(* PLC project Controller_Project, Sphere_UseCases Controller_Project 1.0 *)
(* stored: creationDateTime 2025-09-25T18:23:17, modificationDateTime 2025-09-25T18:23:17 *)

TYPE HMI_UDT : STRUCT
  Start_PB : BOOL;
  Stop_PB : BOOL;
  Start_Active : BOOL;
  Stop_Active : BOOL;
END_STRUCT;
END_TYPE

TYPE P1_UDT : STRUCT
  RW_Tank_tnk_lvl : REAL;
  RW_Pump_flow : REAL;
  RW_Tank_PR_Valve_sts : BOOL;
  RW_Tank_P6B_Valve_sts : BOOL;
  RW_Tank_P_Valve_sts : BOOL;
  RW_Pump_sts : BOOL;
  RW_Pump_fault : BOOL;
  RW_Pump : REAL;
  RW_Tank_PR_Valve : BOOL;
  RW_Tank_P_Valve : BOOL;
  RW_Pump_start : BOOL;
  RW_Pump_stop : BOOL;
  RW_Tank_P6B_Valve : BOOL;
END_STRUCT;
END_TYPE

TYPE P2_UDT : STRUCT
  ChemTreat_NaCl_Tank_tnk_lvl : REAL;
  ChemTreat_NaOCl_Tank_tnk_lvl : REAL;
  ChemTreat_HCl_Tank_tnk_lvl : REAL;
  ChemTreat_NaCl_Tank_Valve_sts : BOOL;
  ChemTreat_NaOCl_Tank_Valve_sts : BOOL;
  ChemTreat_HCl_Tank_Valve_sts : BOOL;
  ChemTreat_NaCl_Tank_Valve : BOOL;
  ChemTreat_NaOCl_Tank_Valve : BOOL;
  ChemTreat_HCl_Tank_Valve : BOOL;
END_STRUCT;
END_TYPE

TYPE P3_UDT : STRUCT
  Ultrafiltration_UFFT_Tank_tnk_lvl : REAL;
  Ultrafiltration_UFFT_Tank_Valve_sts : BOOL;
  Ultrafiltration_UF_Drain_Valve_sts : BOOL;
  Ultrafiltration_UF_ROFT_Valve_sts : BOOL;
  Ultrafiltration_UF_BWP_Valve_sts : BOOL;
  Ultrafiltration_UFFT_Tank_Valve : BOOL;
  Ultrafiltration_UF_Drain_Valve : BOOL;
  Ultrafiltration_UF_ROFT_Valve : BOOL;
  Ultrafiltration_UF_BWP_Valve : BOOL;
END_STRUCT;
END_TYPE

TYPE Phases_UDT : STRUCT
  Filling : BOOL;
  Draining : BOOL;
END_STRUCT;
END_TYPE

TYPE RW_tank_AL_UDT : STRUCT
  LL_alarm : BOOL;
  L_alarm : BOOL;
  H_alarm : BOOL;
  HH_alarm : BOOL;
END_STRUCT;
END_TYPE

TYPE System_State_UDT : STRUCT
  IDLE : BOOL;
  START : BOOL;
  RUNNING : BOOL;
  SHUTDOWN : BOOL;
  Permissives : ARRAY[0..31] OF BOOL;
  Permissives_Ready : BOOL;
END_STRUCT;
END_TYPE

TYPE SYS_MESSAGES : STRUCT
  ProgramScanTime : DINT;
  AvailableMemory : REAL;
  ControllerStatus : SINT;
  ScanTime : REAL;
END_STRUCT;
END_TYPE

PROGRAM MainProgram
  VAR_INPUT
    dbg_Alarms_ZZZZZZZZZZRW_tank_AL0 : SINT;
    dbg_Alarms_LL_alarm : BOOL;
    dbg_Alarms_L_alarm : BOOL;
    dbg_Alarms_H_alarm : BOOL;
    dbg_Alarms_HH_alarm : BOOL;
    dbg_GSV_Message_ProgramScanTime : DINT;
    dbg_GSV_Message_AvailableMemory : REAL;
    dbg_GSV_Message_ControllerStatus : SINT;
    dbg_GSV_Message_ScanTime : REAL;
    dbg_HMI_ZZZZZZZZZZUDT0 : SINT;
    dbg_HMI_Start_PB : BOOL;
    dbg_HMI_Stop_PB : BOOL;
    dbg_HMI_Start_Active : BOOL;
    dbg_HMI_Stop_Active : BOOL;
    dbg_P1_RW_Tank_tnk_lvl : REAL;
    dbg_P1_RW_Pump_flow : REAL;
    dbg_P1_ZZZZZZZZZZP1_UDT2 : SINT;
    dbg_P1_RW_Tank_PR_Valve_sts : BOOL;
    dbg_P1_RW_Tank_P6B_Valve_sts : BOOL;
    dbg_P1_RW_Tank_P_Valve_sts : BOOL;
    dbg_P1_RW_Pump_sts : BOOL;
    dbg_P1_RW_Pump_fault : BOOL;
    dbg_P1_RW_Pump : REAL;
    dbg_P1_ZZZZZZZZZZP1_UDT9 : SINT;
    dbg_P1_RW_Tank_PR_Valve : BOOL;
    dbg_P1_RW_Tank_P_Valve : BOOL;
    dbg_P1_RW_Pump_start : BOOL;
    dbg_P1_RW_Pump_stop : BOOL;
    dbg_P1_RW_Tank_P6B_Valve : BOOL;
    dbg_P1_SYS_ZZZZZZZZZZSystem_Sta0 : SINT;
    dbg_P1_SYS_IDLE : BOOL;
    dbg_P1_SYS_START : BOOL;
    dbg_P1_SYS_RUNNING : BOOL;
    dbg_P1_SYS_SHUTDOWN : BOOL;
    dbg_P1_SYS_Permissives : ARRAY[0..31] OF BOOL;
    dbg_P1_SYS_ZZZZZZZZZZSystem_Sta6 : SINT;
    dbg_P1_SYS_Permissives_Ready : BOOL;
    dbg_P2_ChemTreat_NaCl_Tank_tnk_lvl : REAL;
    dbg_P2_ChemTreat_NaOCl_Tank_tnk_lvl : REAL;
    dbg_P2_ChemTreat_HCl_Tank_tnk_lvl : REAL;
    dbg_P2_ZZZZZZZZZZP2_UDT3 : SINT;
    dbg_P2_ChemTreat_NaCl_Tank_Valve_sts : BOOL;
    dbg_P2_ChemTreat_NaOCl_Tank_Valve_sts : BOOL;
    dbg_P2_ChemTreat_HCl_Tank_Valve_sts : BOOL;
    dbg_P2_ChemTreat_NaCl_Tank_Valve : BOOL;
    dbg_P2_ChemTreat_NaOCl_Tank_Valve : BOOL;
    dbg_P2_ChemTreat_HCl_Tank_Valve : BOOL;
    dbg_P3_Ultrafiltration_UFFT_Tank_tnk_lvl : REAL;
    dbg_P3_ZZZZZZZZZZP3_UDT1 : SINT;
    dbg_P3_Ultrafiltration_UFFT_Tank_Valve_sts : BOOL;
    dbg_P3_Ultrafiltration_UF_Drain_Valve_sts : BOOL;
    dbg_P3_Ultrafiltration_UF_ROFT_Valve_sts : BOOL;
    dbg_P3_Ultrafiltration_UF_BWP_Valve_sts : BOOL;
    dbg_P3_Ultrafiltration_UFFT_Tank_Valve : BOOL;
    dbg_P3_Ultrafiltration_UF_Drain_Valve : BOOL;
    dbg_P3_Ultrafiltration_UF_ROFT_Valve : BOOL;
    dbg_P3_Ultrafiltration_UF_BWP_Valve : BOOL;
    di_2_0 AT %IX2.0 : BOOL;
    di_2_1 AT %IX2.1 : BOOL;
    di_2_10 AT %IX2.10 : BOOL;
    di_2_11 AT %IX2.11 : BOOL;
    di_2_2 AT %IX2.2 : BOOL;
    di_2_3 AT %IX2.3 : BOOL;
    di_2_4 AT %IX2.4 : BOOL;
    di_2_5 AT %IX2.5 : BOOL;
    di_2_6 AT %IX2.6 : BOOL;
    di_2_8 AT %IX2.8 : BOOL;
    di_2_9 AT %IX2.9 : BOOL;
    ai_7_0 AT %IW70 : REAL;
    di_7_ch0halarm AT %IX7.0 : BOOL;
    di_7_ch0hhalarm AT %IX7.0 : BOOL;
    di_7_ch0lalarm AT %IX7.0 : BOOL;
    di_7_ch0llalarm AT %IX7.0 : BOOL;
    ai_7_1 AT %IW71 : REAL;
    ai_7_2 AT %IW72 : REAL;
    ai_7_3 AT %IW73 : REAL;
    ai_7_4 AT %IW74 : REAL;
    ai_7_5 AT %IW75 : REAL;
  END_VAR
  VAR_OUTPUT
    ao_10_0 AT %QW100 : REAL;
    do_5_0 AT %QX5.0 : BOOL;
    do_5_1 AT %QX5.1 : BOOL;
    do_5_10 AT %QX5.10 : BOOL;
    do_5_11 AT %QX5.11 : BOOL;
    do_5_2 AT %QX5.2 : BOOL;
    do_5_3 AT %QX5.3 : BOOL;
    do_5_4 AT %QX5.4 : BOOL;
    do_5_5 AT %QX5.5 : BOOL;
    do_5_6 AT %QX5.6 : BOOL;
    do_5_7 AT %QX5.7 : BOOL;
    do_5_8 AT %QX5.8 : BOOL;
    do_5_9 AT %QX5.9 : BOOL;
  END_VAR

            (* IO_setup *)
(* P1 Analog Input *)
dbg_P1_RW_Tank_tnk_lvl := ai_7_0;
dbg_P1_RW_Pump_flow := ai_7_1;
(* P1 Digital Input *)
dbg_P1_RW_Tank_PR_Valve_sts := di_2_0;
dbg_P1_RW_Tank_P6B_Valve_sts := di_2_1;
dbg_P1_RW_Tank_P_Valve_sts := di_2_2;
dbg_P1_RW_Pump_sts := di_2_3;
dbg_P1_RW_Pump_fault := di_2_4;
(* P1 Analog Output *)
dbg_P1_RW_Pump := ao_10_0;
(* Digital Output *)
dbg_P1_RW_Tank_PR_Valve := do_5_0;
dbg_P1_RW_Tank_P6B_Valve := do_5_1;
dbg_P1_RW_Tank_P_Valve := do_5_2;
dbg_P1_RW_Pump_start := do_5_3;
dbg_P1_RW_Pump_stop := do_5_4;
(* P1 raw water tank alarms *)
dbg_Alarms_LL_alarm := di_7_ch0llalarm;
dbg_Alarms_L_alarm := di_7_ch0lalarm;
dbg_Alarms_H_alarm := di_7_ch0halarm;
dbg_Alarms_HH_alarm := di_7_ch0hhalarm;
(* P2 Analog Input *)
dbg_P2_ChemTreat_NaCl_Tank_tnk_lvl := ai_7_2;
dbg_P2_ChemTreat_NaOCl_Tank_tnk_lvl := ai_7_3;
dbg_P2_ChemTreat_HCl_Tank_tnk_lvl := ai_7_4;
(* P2 Digital Input *)
dbg_P2_ChemTreat_NaCl_Tank_Valve_sts := di_2_5;
dbg_P2_ChemTreat_NaOCl_Tank_Valve_sts := di_2_6;
(* P2 Analog Output *)
(* NONE *)
(* P2 Digital Output *)
dbg_P2_ChemTreat_NaCl_Tank_Valve := do_5_5;
dbg_P2_ChemTreat_NaOCl_Tank_Valve := do_5_6;
dbg_P2_ChemTreat_HCl_Tank_Valve := do_5_7;
(* P3 Analog Input *)
dbg_P3_Ultrafiltration_UFFT_Tank_tnk_lvl := ai_7_5;
(* P3 Digital Input *)
dbg_P3_Ultrafiltration_UFFT_Tank_Valve_sts := di_2_8;
dbg_P3_Ultrafiltration_UF_Drain_Valve_sts := di_2_9;
dbg_P3_Ultrafiltration_UF_Drain_Valve_sts := di_2_10;
dbg_P3_Ultrafiltration_UF_BWP_Valve_sts := di_2_11;
(* P3 Analog Output *)
(* none *)
(* P3 Digital Output *)
dbg_P3_Ultrafiltration_UFFT_Tank_Valve := do_5_8;
dbg_P3_Ultrafiltration_UF_Drain_Valve := do_5_9;
dbg_P3_Ultrafiltration_UF_ROFT_Valve := do_5_10;
dbg_P3_Ultrafiltration_UF_BWP_Valve := do_5_11;

(* Raw_water_control *)
if dbg_P1_RW_Tank_tnk_lvl = 250.0 and dbg_P1_SYS_RUNNING then
dbg_P1_RW_Pump_stop := True;
dbg_P1_RW_Pump_start := False; (* send the outputs *)
dbg_Alarms_LL_alarm := True;
(* if the level is at 500 or lower than 500 open the valve *)
elsif dbg_P1_RW_Tank_tnk_lvl <= 500.0 and dbg_P1_SYS_RUNNING then
(* output to turn the valve open *)
dbg_P1_RW_Tank_PR_Valve := True;
dbg_Alarms_L_alarm := True;
(* if level is at 800 *)
elsif  dbg_P1_RW_Tank_tnk_lvl = 800.0 and dbg_P1_SYS_RUNNING then
dbg_P1_RW_Tank_PR_Valve := False; (* close the valve *)
dbg_Alarms_H_alarm := True;
elsif dbg_P1_RW_Tank_tnk_lvl = 1200.0 and dbg_P1_SYS_RUNNING then
dbg_Alarms_HH_alarm := True; (* if the tank is higher than or equal to 1200 set the high high alarm *)
end_if;

(* Raw_water_pump *)
if dbg_P3_Ultrafiltration_UFFT_Tank_tnk_lvl = 800.0 AND dbg_P1_SYS_RUNNING then
(* start the pump and open the valve from the other tank *)
dbg_P1_RW_Tank_P_Valve := True;
dbg_P1_RW_Pump_start := True;
dbg_P1_RW_Pump_stop := False;
elsif dbg_P3_Ultrafiltration_UFFT_Tank_tnk_lvl = 1000.0 AND dbg_P1_SYS_RUNNING then
(* stop the pump and close the valve *)
dbg_P1_RW_Tank_P_Valve := False;
dbg_P1_RW_Pump_stop := True;
dbg_P1_RW_Pump_start := False;
end_if;

(* State_change *)
if not dbg_HMI_Start_Active AND not dbg_HMI_Stop_Active then
(* if start and stop is not pressed go to idle *)
dbg_P1_SYS_IDLE := True;
dbg_P1_SYS_START := False;
dbg_P1_SYS_RUNNING := False;
dbg_P1_SYS_SHUTDOWN := False;
elsif  dbg_HMI_Start_Active AND not dbg_HMI_Stop_Active then
(* if the start pb and stop is not pressed then change the state of process one to starting *)
dbg_P1_SYS_IDLE := False;
dbg_P1_SYS_START := True;
dbg_P1_SYS_RUNNING := False;
dbg_P1_SYS_SHUTDOWN := False;
(* if the tank level is greater than 250 at the start and UFFT is less than a 1000 we can start *)
(* then and all permissves cond together into one tag so we know the plant is ready to start *)
dbg_P1_SYS_Permissives_Ready := dbg_P1_SYS_Permissives[0] AND dbg_P1_SYS_Permissives[1];
elsif dbg_HMI_Start_Active AND dbg_P1_SYS_Permissives_Ready then
(* if the start was pressed and permissives are ready start running Process one *)
dbg_P1_SYS_IDLE := False;
dbg_P1_SYS_START := False;
dbg_P1_SYS_RUNNING := True;
dbg_P1_SYS_SHUTDOWN := False;
elsif dbg_HMI_Stop_Active then
(* if the stop button is pressed then go to shutdown state *)
dbg_P1_SYS_IDLE := False;
dbg_P1_SYS_START := False;
dbg_P1_SYS_RUNNING := False;
dbg_P1_SYS_SHUTDOWN := True;
(* set all permissives to false *)
dbg_P1_SYS_Permissives_Ready := False;
end_if;

          
END_PROGRAM

CONFIGURATION config
  VAR_GLOBAL
    ao_10_0 AT %QW100 : REAL;  (* Rockwell: Local:10:O.Ch0Data *)
    di_2_0 AT %IX2.0 : BOOL;  (* Rockwell: Local:2:I.Data.0 *)
    di_2_1 AT %IX2.1 : BOOL;  (* Rockwell: Local:2:I.Data.1 *)
    di_2_10 AT %IX2.10 : BOOL;  (* Rockwell: Local:2:I.Data.10 *)
    di_2_11 AT %IX2.11 : BOOL;  (* Rockwell: Local:2:I.Data.11 *)
    di_2_2 AT %IX2.2 : BOOL;  (* Rockwell: Local:2:I.Data.2 *)
    di_2_3 AT %IX2.3 : BOOL;  (* Rockwell: Local:2:I.Data.3 *)
    di_2_4 AT %IX2.4 : BOOL;  (* Rockwell: Local:2:I.Data.4 *)
    di_2_5 AT %IX2.5 : BOOL;  (* Rockwell: Local:2:I.Data.5 *)
    di_2_6 AT %IX2.6 : BOOL;  (* Rockwell: Local:2:I.Data.6 *)
    di_2_8 AT %IX2.8 : BOOL;  (* Rockwell: Local:2:I.Data.8 *)
    di_2_9 AT %IX2.9 : BOOL;  (* Rockwell: Local:2:I.Data.9 *)
    do_5_0 AT %QX5.0 : BOOL;  (* Rockwell: Local:5:O.Data.0 *)
    do_5_1 AT %QX5.1 : BOOL;  (* Rockwell: Local:5:O.Data.1 *)
    do_5_10 AT %QX5.10 : BOOL;  (* Rockwell: Local:5:O.Data.10 *)
    do_5_11 AT %QX5.11 : BOOL;  (* Rockwell: Local:5:O.Data.11 *)
    do_5_2 AT %QX5.2 : BOOL;  (* Rockwell: Local:5:O.Data.2 *)
    do_5_3 AT %QX5.3 : BOOL;  (* Rockwell: Local:5:O.Data.3 *)
    do_5_4 AT %QX5.4 : BOOL;  (* Rockwell: Local:5:O.Data.4 *)
    do_5_5 AT %QX5.5 : BOOL;  (* Rockwell: Local:5:O.Data.5 *)
    do_5_6 AT %QX5.6 : BOOL;  (* Rockwell: Local:5:O.Data.6 *)
    do_5_7 AT %QX5.7 : BOOL;  (* Rockwell: Local:5:O.Data.7 *)
    do_5_8 AT %QX5.8 : BOOL;  (* Rockwell: Local:5:O.Data.8 *)
    do_5_9 AT %QX5.9 : BOOL;  (* Rockwell: Local:5:O.Data.9 *)
    ai_7_0 AT %IW70 : REAL;  (* Rockwell: Local:7:I.Ch0Data *)
    di_7_ch0halarm AT %IX7.0 : BOOL;  (* Rockwell: Local:7:I.Ch0HAlarm *)
    di_7_ch0hhalarm AT %IX7.0 : BOOL;  (* Rockwell: Local:7:I.Ch0HHAlarm *)
    di_7_ch0lalarm AT %IX7.0 : BOOL;  (* Rockwell: Local:7:I.Ch0LAlarm *)
    di_7_ch0llalarm AT %IX7.0 : BOOL;  (* Rockwell: Local:7:I.Ch0LLAlarm *)
    ai_7_1 AT %IW71 : REAL;  (* Rockwell: Local:7:I.Ch1Data *)
    ai_7_2 AT %IW72 : REAL;  (* Rockwell: Local:7:I.Ch2Data *)
    ai_7_3 AT %IW73 : REAL;  (* Rockwell: Local:7:I.Ch3Data *)
    ai_7_4 AT %IW74 : REAL;  (* Rockwell: Local:7:I.Ch4Data *)
    ai_7_5 AT %IW75 : REAL;  (* Rockwell: Local:7:I.Ch5Data *)
  END_VAR
  RESOURCE res_MainProgram ON PLC
    TASK task_MainProgram(INTERVAL := T#100ms, PRIORITY := 0);
    PROGRAM MainProgram_instance : MainProgram;
  END_RESOURCE
END_CONFIGURATION
